(* Schneider Machine Expert - Basic project A1, file version 2.7.0.0 *)
(* ProjectInformations: Name=Novo projeto *)
(* UserInformations: LastName=foda-se *)

HARDWARE
  Cpu 0: TM221M16R/G
  ModuleExtensionObject 0: TM3DI16/G
  EthernetConfiguration: NetworkName=M221, IpAllocationMode=FixedAddress, IpAddress=0.0.0.0, SubnetMask=0.0.0.0
  SerialLineConfiguration: Baud=Baud19200, Parity=ParityEven, DataBits=DataBits8, StopBits=StopBits1, PhysicalMedium=PhysicalMediumRs485, TransmissionMode=TransmissionModeModbusRtu, SlaveId=1, Addressing=SlaveAddressing
  MastTask: UsePeriodScanMode=false, PeriodScan=100
  FastTask: Period=255
  CpuBehavior: StartingMode=StartAsPreviousState, AutoSaveRamOnEeprom=true, WatchdogPeriod=250

SYMBOLS  (address, symbol, comment, settings)

POU Novo POU  (* Comando Bomba de Água *)
  (* SectionNumber=0 *)

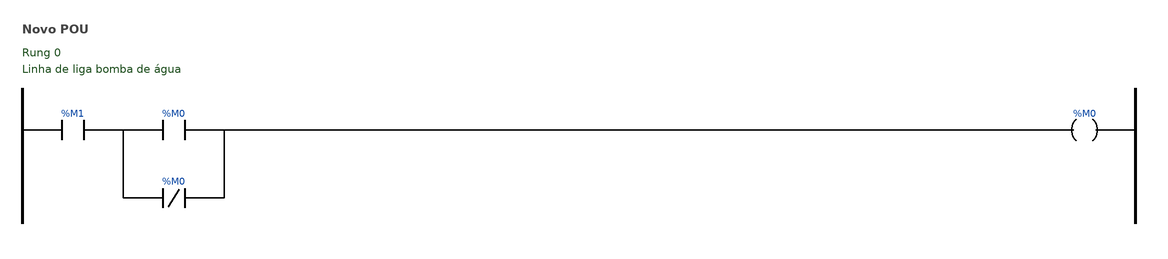

// Rung 0
// Linha de liga bomba de água
  LD %M1
  AND( %M0
  ORN %M0
  )
  ST %M0
  // as ST:
  //   %M0 := %M1 AND (%M0 OR NOT %M0);
